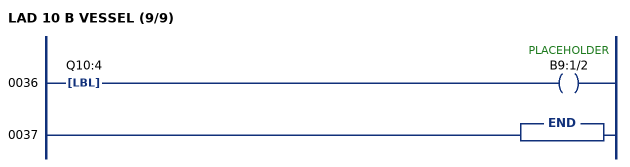
% Rung: 36 %
SOR LBL Q10:4 OTE B9:1/2 EOR
%   B9:1/2  "PLACEHOLDER" %
% Rung: 37 %
SOR END EOR

LADDER 11 "DIGITAL IN"
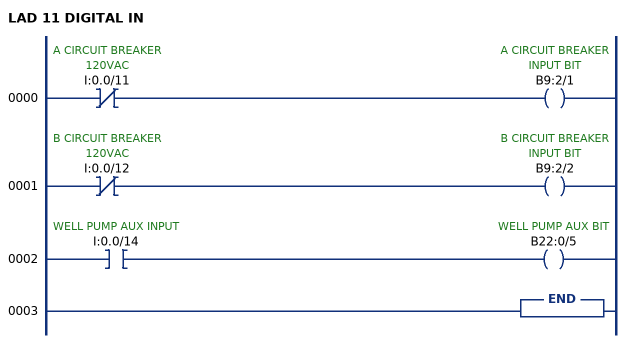
% Rung: 0 %
SOR XIO I:0.0/11 OTE B9:2/1 EOR
%   I:0.0/11  "A CIRCUIT BREAKER 120VAC" %
%   B9:2/1  "A CIRCUIT BREAKER INPUT BIT" %
% Rung: 1 %
SOR XIO I:0.0/12 OTE B9:2/2 EOR
%   I:0.0/12  "B CIRCUIT BREAKER 120VAC" %
%   B9:2/2  "B CIRCUIT BREAKER INPUT BIT" %
% Rung: 2 %
SOR XIC I:0.0/14 OTE B22:0/5 EOR
%   I:0.0/14  "WELL PUMP AUX INPUT" %
%   B22:0/5  "WELL PUMP AUX BIT" %
% Rung: 3 %
SOR END EOR

LADDER 12 "WELL PUMP"
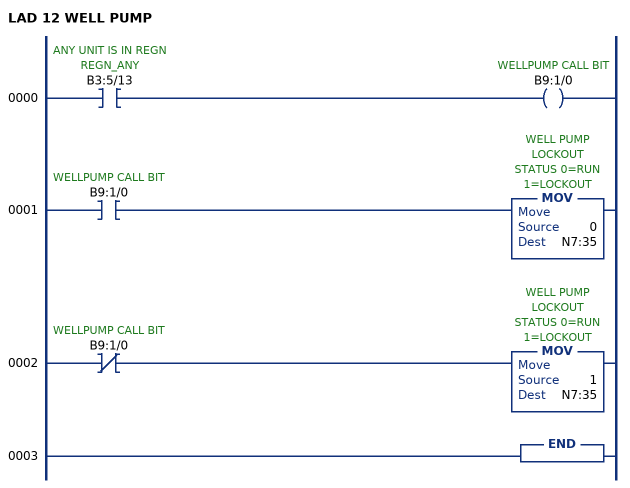
% Rung: 0 %
SOR XIC B3:5/13 OTE B9:1/0 EOR
%   B3:5/13  REGN_ANY  "ANY UNIT IS IN REGN" %
%   B9:1/0  "WELLPUMP CALL BIT" %
% Rung: 1 %
SOR XIC B9:1/0 MOV 0 N7:35 EOR
%   B9:1/0  "WELLPUMP CALL BIT" %
%   N7:35  "WELL PUMP LOCKOUT STATUS 0=RUN 1=LOCKOUT" %
% Rung: 2 %
SOR XIO B9:1/0 MOV 1 N7:35 EOR
%   B9:1/0  "WELLPUMP CALL BIT" %
%   N7:35  "WELL PUMP LOCKOUT STATUS 0=RUN 1=LOCKOUT" %
% Rung: 3 %
SOR END EOR

LADDER 16 "DIGITL OUT"
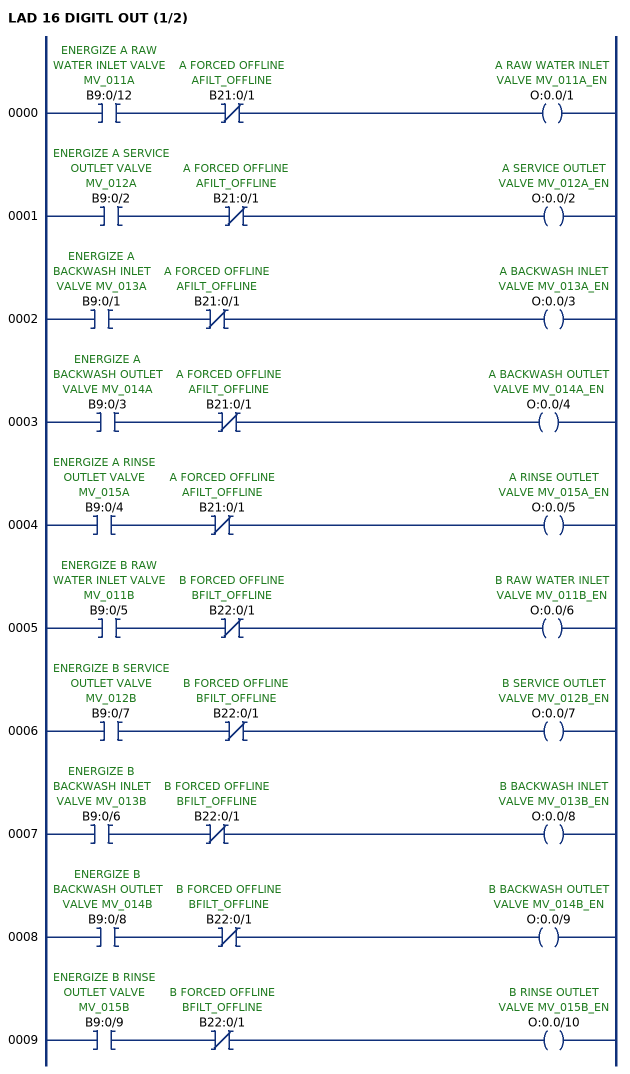
% Rung: 0 %
SOR XIC B9:0/12 XIO B21:0/1 OTE O:0.0/1 EOR
%   B9:0/12  MV_011A  "ENERGIZE A RAW WATER INLET VALVE" %
%   B21:0/1  AFILT_OFFLINE  "A FORCED OFFLINE" %
%   O:0.0/1  MV_011A_EN  "A RAW WATER INLET VALVE" %
% Rung: 1 %
SOR XIC B9:0/2 XIO B21:0/1 OTE O:0.0/2 EOR
%   B9:0/2  MV_012A  "ENERGIZE A SERVICE OUTLET VALVE" %
%   B21:0/1  AFILT_OFFLINE  "A FORCED OFFLINE" %
%   O:0.0/2  MV_012A_EN  "A SERVICE OUTLET VALVE" %
% Rung: 2 %
SOR XIC B9:0/1 XIO B21:0/1 OTE O:0.0/3 EOR
%   B9:0/1  MV_013A  "ENERGIZE A BACKWASH INLET VALVE" %
%   B21:0/1  AFILT_OFFLINE  "A FORCED OFFLINE" %
%   O:0.0/3  MV_013A_EN  "A BACKWASH INLET VALVE" %
% Rung: 3 %
SOR XIC B9:0/3 XIO B21:0/1 OTE O:0.0/4 EOR
%   B9:0/3  MV_014A  "ENERGIZE A BACKWASH OUTLET VALVE" %
%   B21:0/1  AFILT_OFFLINE  "A FORCED OFFLINE" %
%   O:0.0/4  MV_014A_EN  "A BACKWASH OUTLET VALVE" %
% Rung: 4 %
SOR XIC B9:0/4 XIO B21:0/1 OTE O:0.0/5 EOR
%   B9:0/4  MV_015A  "ENERGIZE A RINSE OUTLET VALVE" %
%   B21:0/1  AFILT_OFFLINE  "A FORCED OFFLINE" %
%   O:0.0/5  MV_015A_EN  "A RINSE OUTLET VALVE" %
% Rung: 5 %
SOR XIC B9:0/5 XIO B22:0/1 OTE O:0.0/6 EOR
%   B9:0/5  MV_011B  "ENERGIZE B RAW WATER INLET VALVE" %
%   B22:0/1  BFILT_OFFLINE  "B FORCED OFFLINE" %
%   O:0.0/6  MV_011B_EN  "B RAW WATER INLET VALVE" %
% Rung: 6 %
SOR XIC B9:0/7 XIO B22:0/1 OTE O:0.0/7 EOR
%   B9:0/7  MV_012B  "ENERGIZE B SERVICE OUTLET VALVE" %
%   B22:0/1  BFILT_OFFLINE  "B FORCED OFFLINE" %
%   O:0.0/7  MV_012B_EN  "B SERVICE OUTLET VALVE" %
% Rung: 7 %
SOR XIC B9:0/6 XIO B22:0/1 OTE O:0.0/8 EOR
%   B9:0/6  MV_013B  "ENERGIZE B BACKWASH INLET VALVE" %
%   B22:0/1  BFILT_OFFLINE  "B FORCED OFFLINE" %
%   O:0.0/8  MV_013B_EN  "B BACKWASH INLET VALVE" %
% Rung: 8 %
SOR XIC B9:0/8 XIO B22:0/1 OTE O:0.0/9 EOR
%   B9:0/8  MV_014B  "ENERGIZE B BACKWASH OUTLET VALVE" %
%   B22:0/1  BFILT_OFFLINE  "B FORCED OFFLINE" %
%   O:0.0/9  MV_014B_EN  "B BACKWASH OUTLET VALVE" %
% Rung: 9 %
SOR XIC B9:0/9 XIO B22:0/1 OTE O:0.0/10 EOR
%   B9:0/9  MV_015B  "ENERGIZE B RINSE OUTLET VALVE" %
%   B22:0/1  BFILT_OFFLINE  "B FORCED OFFLINE" %
%   O:0.0/10  MV_015B_EN  "B RINSE OUTLET VALVE" %

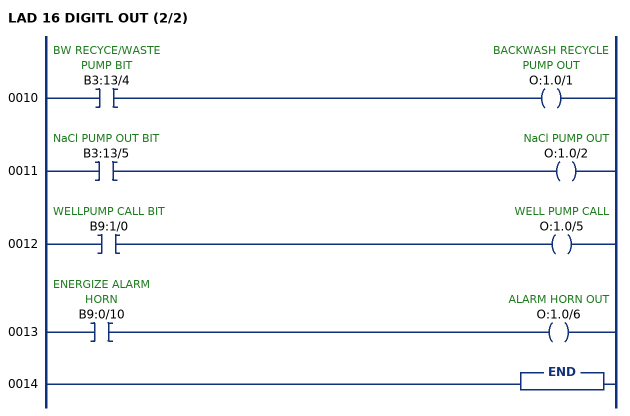
% Rung: 10 %
SOR XIC B3:13/4 OTE O:1.0/1 EOR
%   B3:13/4  "BW RECYCE/WASTE PUMP BIT" %
%   O:1.0/1  "BACKWASH RECYCLE PUMP OUT" %
% Rung: 11 %
SOR XIC B3:13/5 OTE O:1.0/2 EOR
%   B3:13/5  "NaCl PUMP OUT BIT" %
%   O:1.0/2  "NaCl PUMP OUT" %
% Rung: 12 %
SOR XIC B9:1/0 OTE O:1.0/5 EOR
%   B9:1/0  "WELLPUMP CALL BIT" %
%   O:1.0/5  "WELL PUMP CALL" %
% Rung: 13 %
SOR XIC B9:0/10 OTE O:1.0/6 EOR
%   B9:0/10  "ENERGIZE ALARM HORN" %
%   O:1.0/6  "ALARM HORN OUT" %
% Rung: 14 %
SOR END EOR

LADDER 17 "REGEN A"
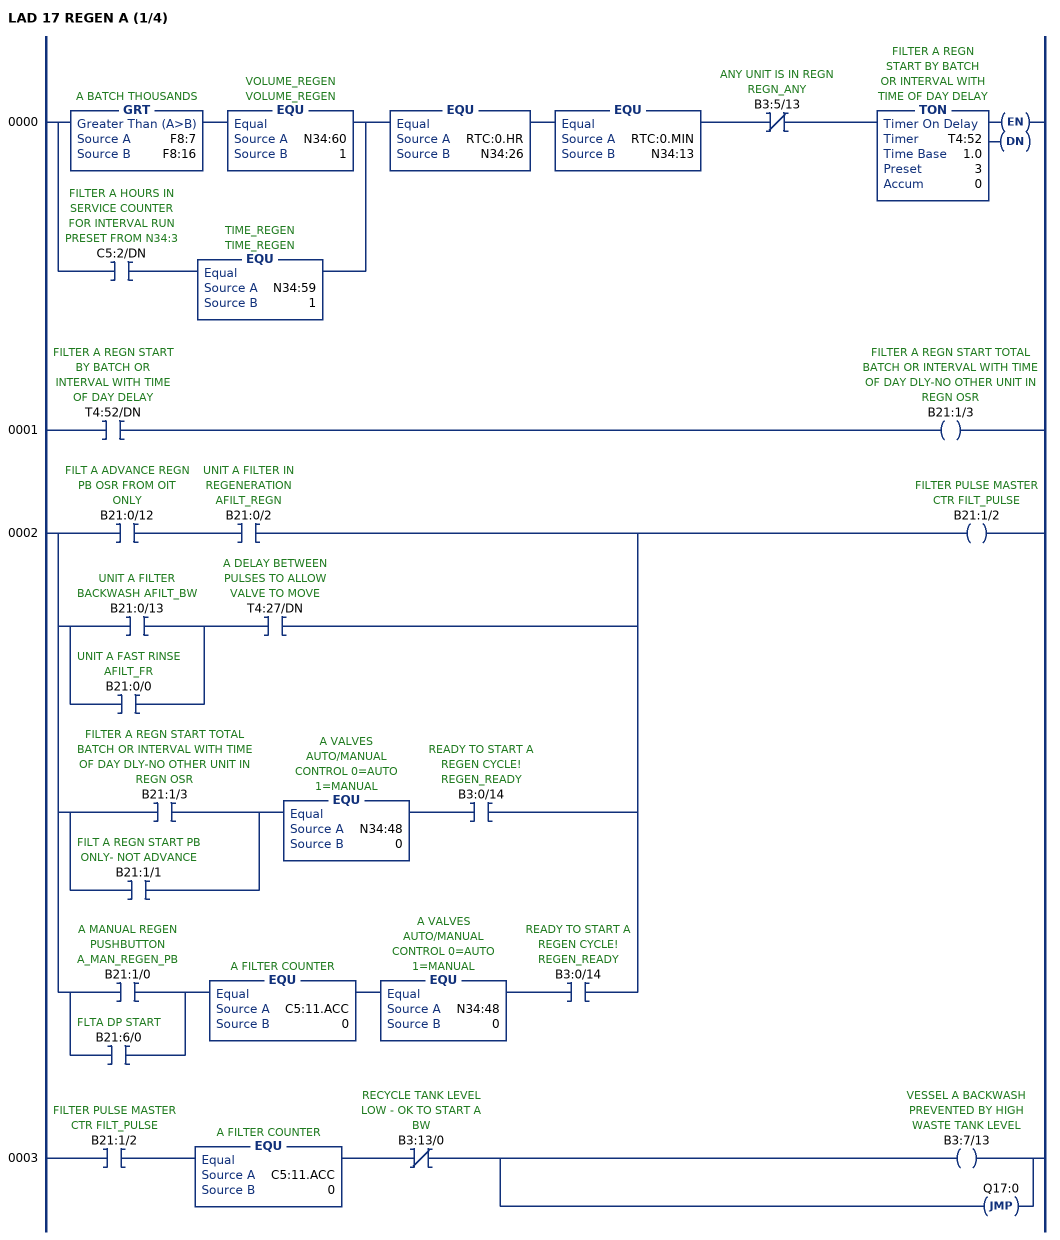
% Rung: 0 %
SOR BST GRT F8:7 F8:16 EQU N34:60 1 NXB XIC C5:2/DN EQU N34:59 1 BND EQU RTC:0.HR N34:26 EQU RTC:0.MIN N34:13 XIO B3:5/13 TON T4:52 1.0 3 0 EOR
%   F8:7  "A BATCH THOUSANDS" %
%   F8:16  T_GAL %
%   N34:60  VOLUME_REGEN  "VOLUME_REGEN" %
%   C5:2  "FILTER A HOURS IN SERVICE COUNTER FOR INTERVAL RUN PRESET FROM N34:3" %
%   N34:59  TIME_REGEN  "TIME_REGEN" %
%   N34:26  "FILTER A HOUR OF DAY TO START SELECT EITHER DUE TO BATCH OR ELAPSED TIME OR DP" %
%   N34:13  "FILTER A MIN OF DAY TO START SELECT EITHER DUE TO BATCH OR ELAPSED TIME" %
%   B3:5/13  REGN_ANY  "ANY UNIT IS IN REGN" %
%   T4:52  "FILTER A REGN START BY BATCH OR INTERVAL WITH TIME OF DAY DELAY" %
% Rung: 1 %
SOR XIC T4:52/DN OTE B21:1/3 EOR
%   T4:52  "FILTER A REGN START BY BATCH OR INTERVAL WITH TIME OF DAY DELAY" %
%   B21:1/3  "FILTER A REGN START TOTAL BATCH OR INTERVAL WITH TIME OF DAY DLY-NO OTHER UNIT IN REGN OSR" %
% Rung: 2 %
SOR BST BST BST XIC B21:0/12 XIC B21:0/2 NXB BST XIC B21:0/13 NXB XIC B21:0/0 BND XIC T4:27/DN BND NXB BST XIC B21:1/3 NXB XIC B21:1/1 BND EQU N34:48 0 XIC B3:0/14 BND NXB BST XIC B21:1/0 NXB XIC B21:6/0 BND EQU C5:11.ACC 0 EQU N34:48 0 XIC B3:0/14 BND OTE B21:1/2 EOR
%   B21:0/12  "FILT A ADVANCE REGN PB OSR FROM OIT ONLY" %
%   B21:0/2  AFILT_REGN  "UNIT A FILTER IN REGENERATION" %
%   B21:0/13  AFILT_BW  "UNIT A FILTER BACKWASH" %
%   B21:0/0  AFILT_FR  "UNIT A FAST RINSE" %
%   T4:27  "A DELAY BETWEEN PULSES TO ALLOW VALVE TO MOVE" %
%   B21:1/3  "FILTER A REGN START TOTAL BATCH OR INTERVAL WITH TIME OF DAY DLY-NO OTHER UNIT IN REGN OSR" %
%   B21:1/1  "FILT A REGN START PB ONLY- NOT ADVANCE" %
%   N34:48  "A VALVES AUTO/MANUAL CONTROL 0=AUTO 1=MANUAL" %
%   B3:0/14  REGEN_READY  "READY TO START A REGEN CYCLE!" %
%   B21:1/0  A_MAN_REGEN_PB  "A MANUAL REGEN PUSHBUTTON" %
%   B21:6/0  "FLTA DP START" %
%   C5:11.ACC  "A FILTER COUNTER" %
%   B21:1/2  FILT_PULSE  "FILTER PULSE MASTER CTR" %
% Rung: 3 %
SOR XIC B21:1/2 EQU C5:11.ACC 0 XIO B3:13/0 BST OTE B3:7/13 NXB JMP Q17:0 BND EOR
%   B21:1/2  FILT_PULSE  "FILTER PULSE MASTER CTR" %
%   C5:11.ACC  "A FILTER COUNTER" %
%   B3:13/0  "RECYCLE TANK LEVEL LOW - OK TO START A BW" %
%   B3:7/13  "VESSEL A BACKWASH PREVENTED BY HIGH WASTE TANK LEVEL" %

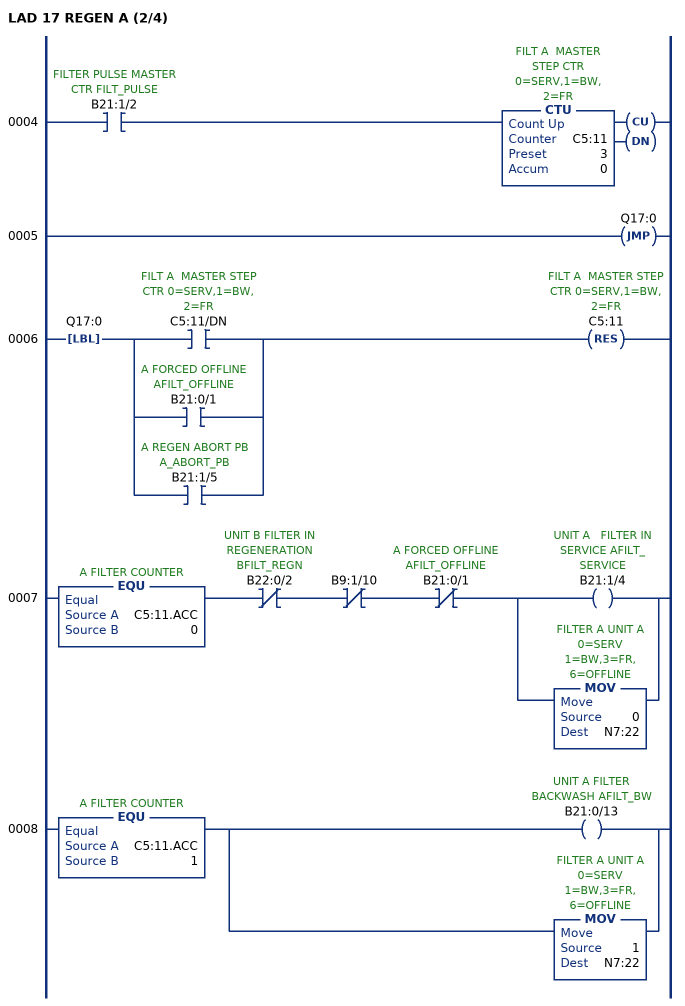
% Rung: 4 %
SOR XIC B21:1/2 CTU C5:11 3 0 EOR
%   B21:1/2  FILT_PULSE  "FILTER PULSE MASTER CTR" %
%   C5:11  "FILT A  MASTER STEP CTR 0=SERV,1=BW,2=FR" %
% Rung: 5 %
SOR JMP Q17:0 EOR
% Rung: 6 %
SOR LBL Q17:0 BST XIC C5:11/DN NXB XIC B21:0/1 NXB XIC B21:1/5 BND RES C5:11 EOR
%   C5:11  "FILT A  MASTER STEP CTR 0=SERV,1=BW,2=FR" %
%   B21:0/1  AFILT_OFFLINE  "A FORCED OFFLINE" %
%   B21:1/5  A_ABORT_PB  "A REGEN ABORT PB" %
% Rung: 7 %
SOR EQU C5:11.ACC 0 XIO B22:0/2 XIO B9:1/10 XIO B21:0/1 BST OTE B21:1/4 NXB MOV 0 N7:22 BND EOR
%   C5:11.ACC  "A FILTER COUNTER" %
%   B22:0/2  BFILT_REGN  "UNIT B FILTER IN REGENERATION" %
%   B21:0/1  AFILT_OFFLINE  "A FORCED OFFLINE" %
%   B21:1/4  AFILT_SERVICE  "UNIT A   FILTER IN SERVICE" %
%   N7:22  "FILTER A UNIT A 0=SERV 1=BW,3=FR,6=OFFLINE" %
% Rung: 8 %
SOR EQU C5:11.ACC 1 BST OTE B21:0/13 NXB MOV 1 N7:22 BND EOR
%   C5:11.ACC  "A FILTER COUNTER" %
%   B21:0/13  AFILT_BW  "UNIT A FILTER BACKWASH" %
%   N7:22  "FILTER A UNIT A 0=SERV 1=BW,3=FR,6=OFFLINE" %

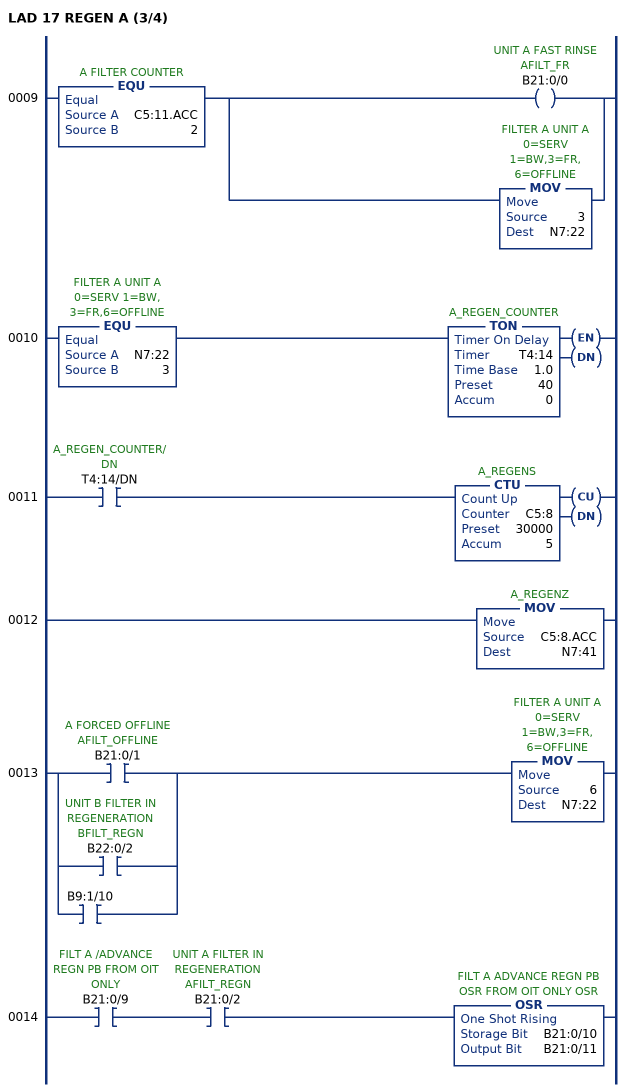
% Rung: 9 %
SOR EQU C5:11.ACC 2 BST OTE B21:0/0 NXB MOV 3 N7:22 BND EOR
%   C5:11.ACC  "A FILTER COUNTER" %
%   B21:0/0  AFILT_FR  "UNIT A FAST RINSE" %
%   N7:22  "FILTER A UNIT A 0=SERV 1=BW,3=FR,6=OFFLINE" %
% Rung: 10 %
SOR EQU N7:22 3 TON T4:14 1.0 40 0 EOR
%   N7:22  "FILTER A UNIT A 0=SERV 1=BW,3=FR,6=OFFLINE" %
%   T4:14  A_REGEN_COUNTER %
% Rung: 11 %
SOR XIC T4:14/DN CTU C5:8 30000 5 EOR
%   T4:14  A_REGEN_COUNTER %
%   C5:8  "A_REGENS" %
% Rung: 12 %
SOR MOV C5:8.ACC N7:41 EOR
%   C5:8  "A_REGENS" %
%   N7:41  A_REGENZ %
% Rung: 13 %
SOR BST XIC B21:0/1 NXB XIC B22:0/2 NXB XIC B9:1/10 BND MOV 6 N7:22 EOR
%   B21:0/1  AFILT_OFFLINE  "A FORCED OFFLINE" %
%   B22:0/2  BFILT_REGN  "UNIT B FILTER IN REGENERATION" %
%   N7:22  "FILTER A UNIT A 0=SERV 1=BW,3=FR,6=OFFLINE" %
% Rung: 14 %
SOR XIC B21:0/9 XIC B21:0/2 OSR B21:0/10 B21:0/11 EOR
%   B21:0/9  "FILT A /ADVANCE REGN PB FROM OIT ONLY" %
%   B21:0/2  AFILT_REGN  "UNIT A FILTER IN REGENERATION" %
%   B21:0/10  "FILT A ADVANCE REGN PB OSR FROM OIT ONLY OSR" %
%   B21:0/11  "FILT A START/ADVANCE REGN PB OSR FROM OIT ONLY OSR" %

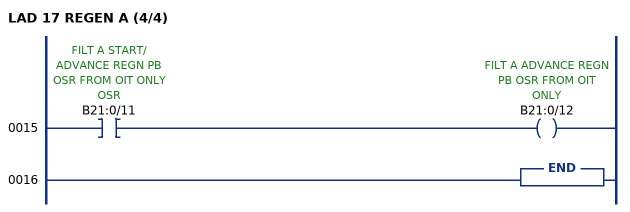
% Rung: 15 %
SOR XIC B21:0/11 OTE B21:0/12 EOR
%   B21:0/11  "FILT A START/ADVANCE REGN PB OSR FROM OIT ONLY OSR" %
%   B21:0/12  "FILT A ADVANCE REGN PB OSR FROM OIT ONLY" %
% Rung: 16 %
SOR END EOR

LADDER 18 "REGEN B"
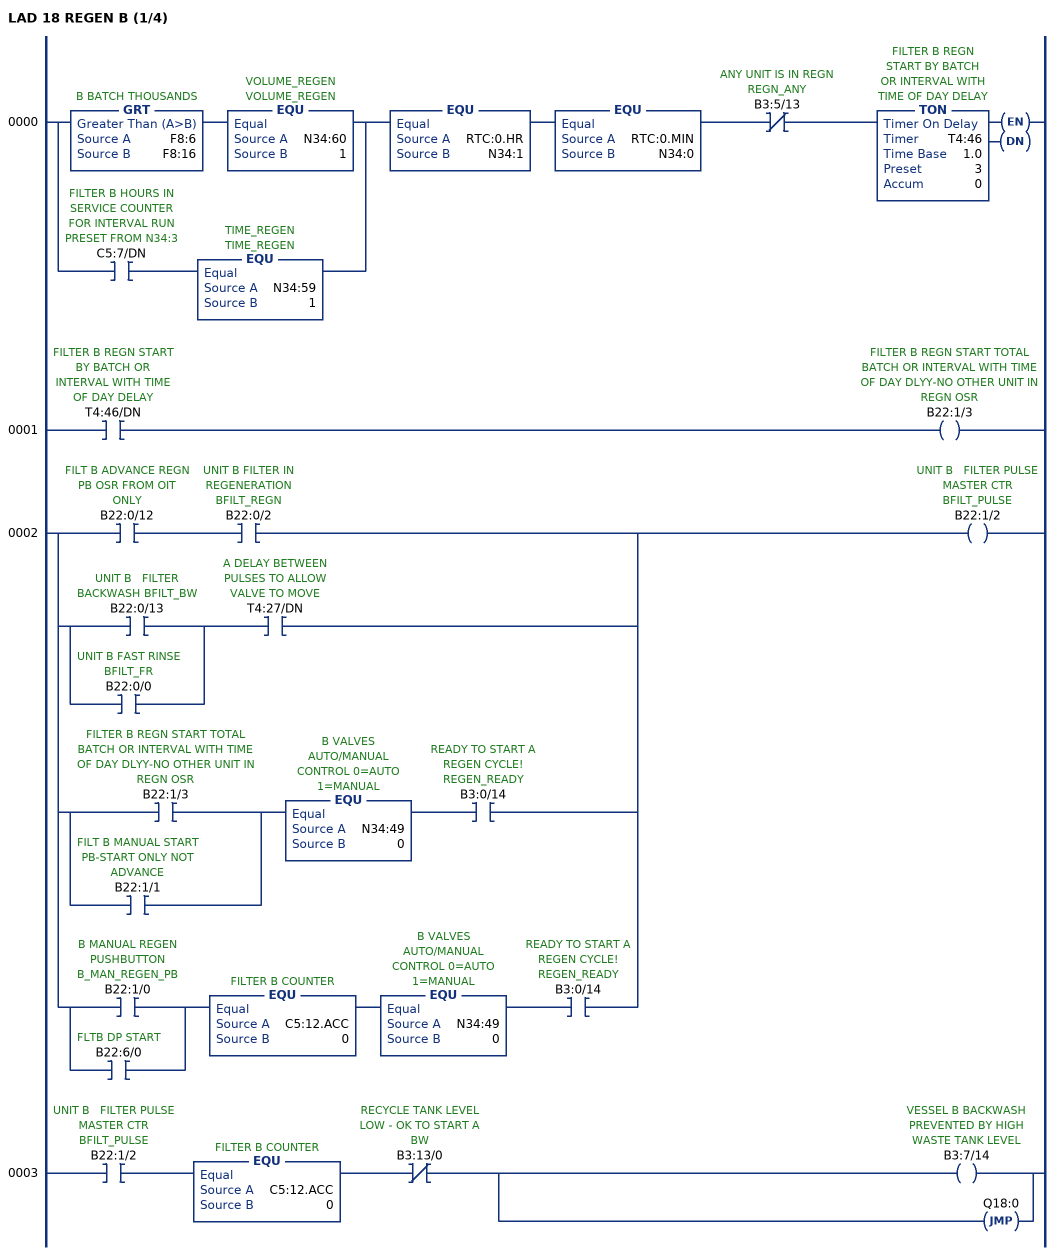
% Rung: 0 %
SOR BST GRT F8:6 F8:16 EQU N34:60 1 NXB XIC C5:7/DN EQU N34:59 1 BND EQU RTC:0.HR N34:1 EQU RTC:0.MIN N34:0 XIO B3:5/13 TON T4:46 1.0 3 0 EOR
%   F8:6  "B BATCH THOUSANDS" %
%   F8:16  T_GAL %
%   N34:60  VOLUME_REGEN  "VOLUME_REGEN" %
%   C5:7  "FILTER B HOURS IN SERVICE COUNTER FOR INTERVAL RUN PRESET FROM N34:3" %
%   N34:59  TIME_REGEN  "TIME_REGEN" %
%   N34:1  "FILTER B HOUR OF DAY TO START SELECT EITHER DUE TO BATCH OR ELAPSED TIME OR DP" %
%   N34:0  "FILTER B MIN OF DAY TO START SELECT EITHER DUE TO BATCH OR ELAPSED TIME" %
%   B3:5/13  REGN_ANY  "ANY UNIT IS IN REGN" %
%   T4:46  "FILTER B REGN START BY BATCH OR INTERVAL WITH TIME OF DAY DELAY" %
% Rung: 1 %
SOR XIC T4:46/DN OTE B22:1/3 EOR
%   T4:46  "FILTER B REGN START BY BATCH OR INTERVAL WITH TIME OF DAY DELAY" %
%   B22:1/3  "FILTER B REGN START TOTAL BATCH OR INTERVAL WITH TIME OF DAY DLYY-NO OTHER UNIT IN REGN OSR" %
% Rung: 2 %
SOR BST BST BST XIC B22:0/12 XIC B22:0/2 NXB BST XIC B22:0/13 NXB XIC B22:0/0 BND XIC T4:27/DN BND NXB BST XIC B22:1/3 NXB XIC B22:1/1 BND EQU N34:49 0 XIC B3:0/14 BND NXB BST XIC B22:1/0 NXB XIC B22:6/0 BND EQU C5:12.ACC 0 EQU N34:49 0 XIC B3:0/14 BND OTE B22:1/2 EOR
%   B22:0/12  "FILT B ADVANCE REGN PB OSR FROM OIT ONLY" %
%   B22:0/2  BFILT_REGN  "UNIT B FILTER IN REGENERATION" %
%   B22:0/13  BFILT_BW  "UNIT B   FILTER BACKWASH" %
%   B22:0/0  BFILT_FR  "UNIT B FAST RINSE" %
%   T4:27  "A DELAY BETWEEN PULSES TO ALLOW VALVE TO MOVE" %
%   B22:1/3  "FILTER B REGN START TOTAL BATCH OR INTERVAL WITH TIME OF DAY DLYY-NO OTHER UNIT IN REGN OSR" %
%   B22:1/1  "FILT B MANUAL START PB-START ONLY NOT ADVANCE" %
%   N34:49  "B VALVES AUTO/MANUAL CONTROL 0=AUTO 1=MANUAL" %
%   B3:0/14  REGEN_READY  "READY TO START A REGEN CYCLE!" %
%   B22:1/0  B_MAN_REGEN_PB  "B MANUAL REGEN PUSHBUTTON" %
%   B22:6/0  "FLTB DP START" %
%   C5:12.ACC  "FILTER B COUNTER" %
%   B22:1/2  BFILT_PULSE  "UNIT B   FILTER PULSE MASTER CTR" %
% Rung: 3 %
SOR XIC B22:1/2 EQU C5:12.ACC 0 XIO B3:13/0 BST OTE B3:7/14 NXB JMP Q18:0 BND EOR
%   B22:1/2  BFILT_PULSE  "UNIT B   FILTER PULSE MASTER CTR" %
%   C5:12.ACC  "FILTER B COUNTER" %
%   B3:13/0  "RECYCLE TANK LEVEL LOW - OK TO START A BW" %
%   B3:7/14  "VESSEL B BACKWASH PREVENTED BY HIGH WASTE TANK LEVEL" %

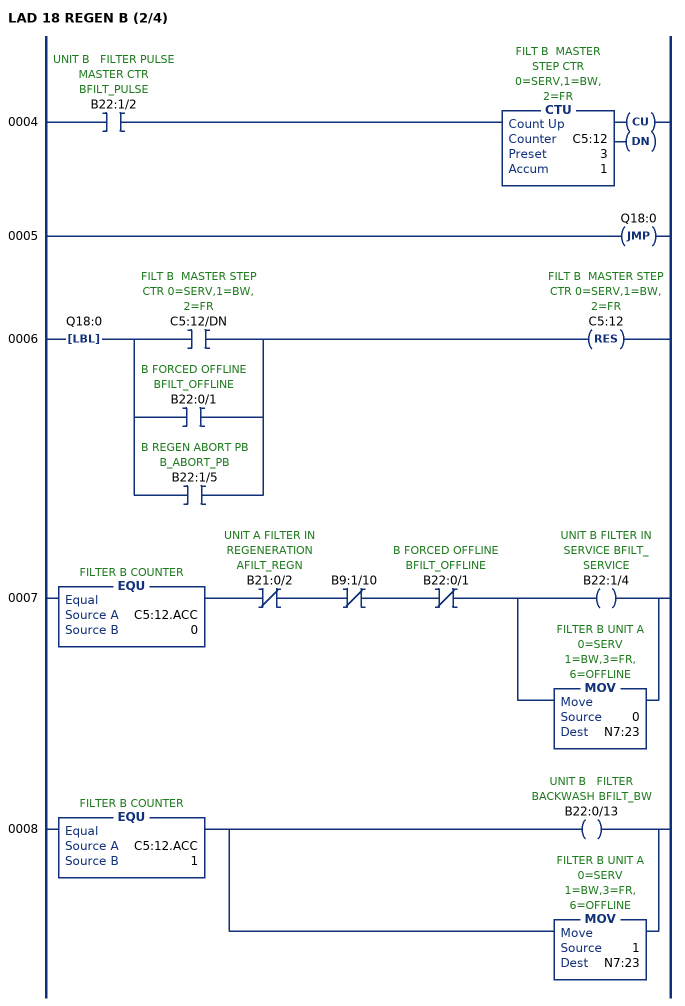
% Rung: 4 %
SOR XIC B22:1/2 CTU C5:12 3 1 EOR
%   B22:1/2  BFILT_PULSE  "UNIT B   FILTER PULSE MASTER CTR" %
%   C5:12  "FILT B  MASTER STEP CTR 0=SERV,1=BW,2=FR" %
% Rung: 5 %
SOR JMP Q18:0 EOR
% Rung: 6 %
SOR LBL Q18:0 BST XIC C5:12/DN NXB XIC B22:0/1 NXB XIC B22:1/5 BND RES C5:12 EOR
%   C5:12  "FILT B  MASTER STEP CTR 0=SERV,1=BW,2=FR" %
%   B22:0/1  BFILT_OFFLINE  "B FORCED OFFLINE" %
%   B22:1/5  B_ABORT_PB  "B REGEN ABORT PB" %
% Rung: 7 %
SOR EQU C5:12.ACC 0 XIO B21:0/2 XIO B9:1/10 XIO B22:0/1 BST OTE B22:1/4 NXB MOV 0 N7:23 BND EOR
%   C5:12.ACC  "FILTER B COUNTER" %
%   B21:0/2  AFILT_REGN  "UNIT A FILTER IN REGENERATION" %
%   B22:0/1  BFILT_OFFLINE  "B FORCED OFFLINE" %
%   B22:1/4  BFILT_SERVICE  "UNIT B FILTER IN SERVICE" %
%   N7:23  "FILTER B UNIT A 0=SERV 1=BW,3=FR,6=OFFLINE" %
% Rung: 8 %
SOR EQU C5:12.ACC 1 BST OTE B22:0/13 NXB MOV 1 N7:23 BND EOR
%   C5:12.ACC  "FILTER B COUNTER" %
%   B22:0/13  BFILT_BW  "UNIT B   FILTER BACKWASH" %
%   N7:23  "FILTER B UNIT A 0=SERV 1=BW,3=FR,6=OFFLINE" %

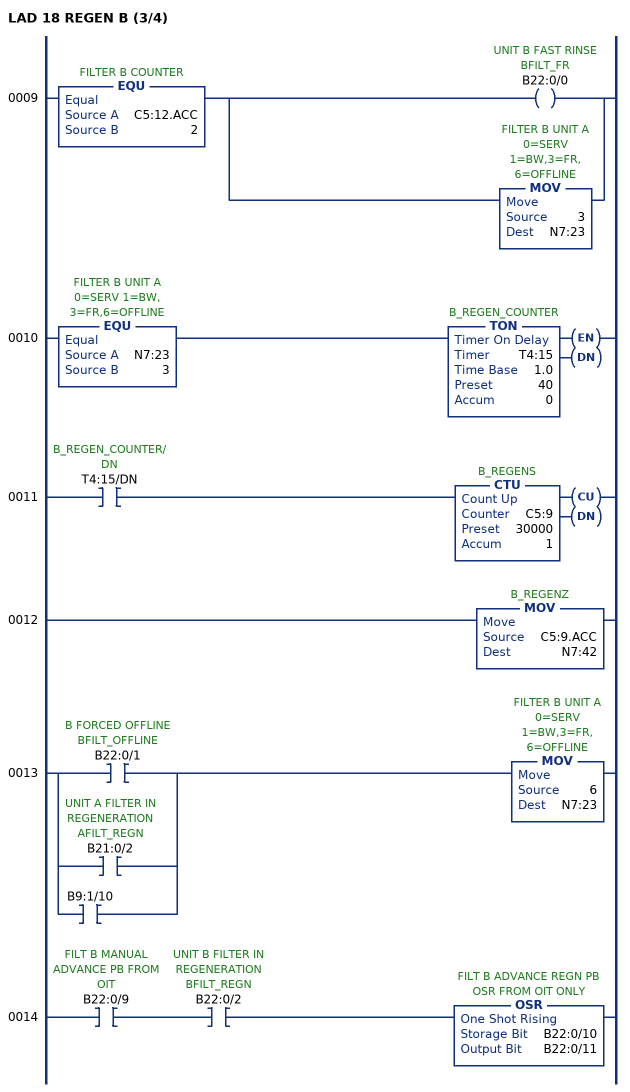
% Rung: 9 %
SOR EQU C5:12.ACC 2 BST OTE B22:0/0 NXB MOV 3 N7:23 BND EOR
%   C5:12.ACC  "FILTER B COUNTER" %
%   B22:0/0  BFILT_FR  "UNIT B FAST RINSE" %
%   N7:23  "FILTER B UNIT A 0=SERV 1=BW,3=FR,6=OFFLINE" %
% Rung: 10 %
SOR EQU N7:23 3 TON T4:15 1.0 40 0 EOR
%   N7:23  "FILTER B UNIT A 0=SERV 1=BW,3=FR,6=OFFLINE" %
%   T4:15  B_REGEN_COUNTER %
% Rung: 11 %
SOR XIC T4:15/DN CTU C5:9 30000 1 EOR
%   T4:15  B_REGEN_COUNTER %
%   C5:9  "B_REGENS" %
% Rung: 12 %
SOR MOV C5:9.ACC N7:42 EOR
%   C5:9  "B_REGENS" %
%   N7:42  B_REGENZ %
% Rung: 13 %
SOR BST XIC B22:0/1 NXB XIC B21:0/2 NXB XIC B9:1/10 BND MOV 6 N7:23 EOR
%   B22:0/1  BFILT_OFFLINE  "B FORCED OFFLINE" %
%   B21:0/2  AFILT_REGN  "UNIT A FILTER IN REGENERATION" %
%   N7:23  "FILTER B UNIT A 0=SERV 1=BW,3=FR,6=OFFLINE" %
% Rung: 14 %
SOR XIC B22:0/9 XIC B22:0/2 OSR B22:0/10 B22:0/11 EOR
%   B22:0/9  "FILT B MANUAL ADVANCE PB FROM OIT" %
%   B22:0/2  BFILT_REGN  "UNIT B FILTER IN REGENERATION" %
%   B22:0/10  "FILT B ADVANCE REGN PB OSR FROM OIT ONLY" %
%   B22:0/11  "FILT B /ADVANCE REGN PB OSR FROM OIT ONLY" %

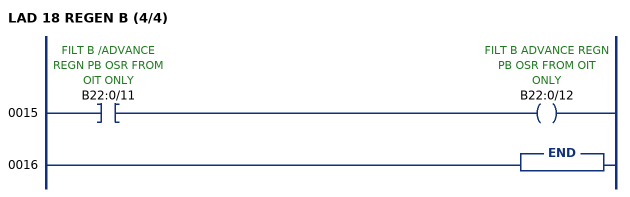
% Rung: 15 %
SOR XIC B22:0/11 OTE B22:0/12 EOR
%   B22:0/11  "FILT B /ADVANCE REGN PB OSR FROM OIT ONLY" %
%   B22:0/12  "FILT B ADVANCE REGN PB OSR FROM OIT ONLY" %
% Rung: 16 %
SOR END EOR

LADDER 19 "RECYCLE"
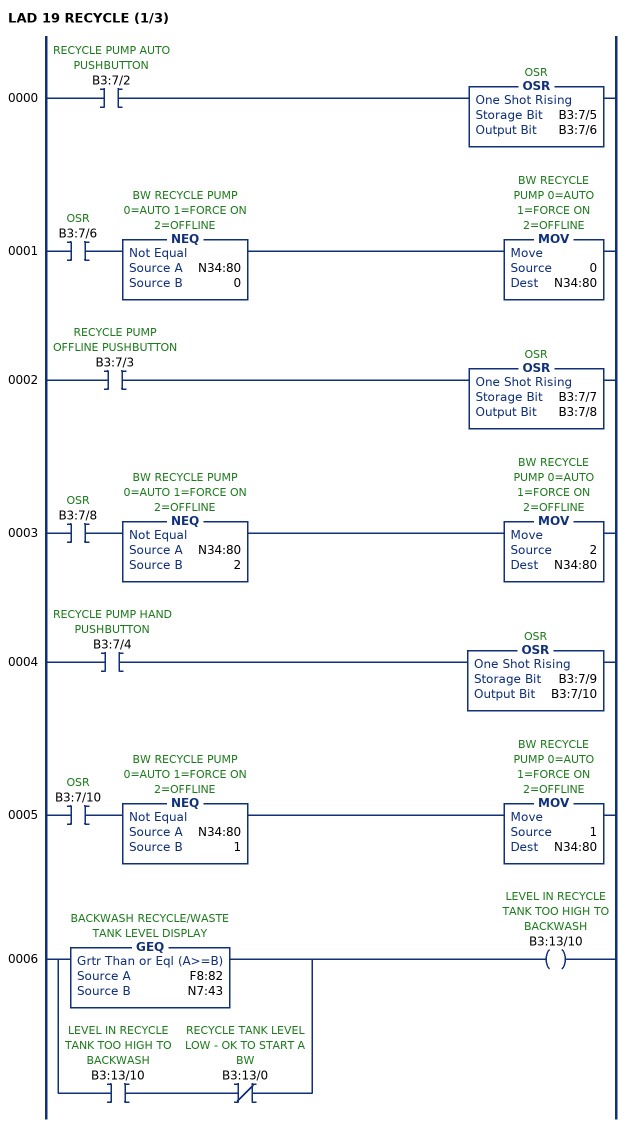
% Rung: 0 %
SOR XIC B3:7/2 OSR B3:7/5 B3:7/6 EOR
%   B3:7/2  "RECYCLE PUMP AUTO PUSHBUTTON" %
%   B3:7/5  "OSR" %
%   B3:7/6  "OSR" %
% Rung: 1 %
SOR XIC B3:7/6 NEQ N34:80 0 MOV 0 N34:80 EOR
%   B3:7/6  "OSR" %
%   N34:80  "BW RECYCLE PUMP 0=AUTO 1=FORCE ON 2=OFFLINE" %
% Rung: 2 %
SOR XIC B3:7/3 OSR B3:7/7 B3:7/8 EOR
%   B3:7/3  "RECYCLE PUMP OFFLINE PUSHBUTTON" %
%   B3:7/7  "OSR" %
%   B3:7/8  "OSR" %
% Rung: 3 %
SOR XIC B3:7/8 NEQ N34:80 2 MOV 2 N34:80 EOR
%   B3:7/8  "OSR" %
%   N34:80  "BW RECYCLE PUMP 0=AUTO 1=FORCE ON 2=OFFLINE" %
% Rung: 4 %
SOR XIC B3:7/4 OSR B3:7/9 B3:7/10 EOR
%   B3:7/4  "RECYCLE PUMP HAND PUSHBUTTON" %
%   B3:7/9  "OSR" %
%   B3:7/10  "OSR" %
% Rung: 5 %
SOR XIC B3:7/10 NEQ N34:80 1 MOV 1 N34:80 EOR
%   B3:7/10  "OSR" %
%   N34:80  "BW RECYCLE PUMP 0=AUTO 1=FORCE ON 2=OFFLINE" %
% Rung: 6 %
SOR BST GEQ F8:82 N7:43 NXB XIC B3:13/10 XIO B3:13/0 BND OTE B3:13/10 EOR
%   F8:82  "BACKWASH RECYCLE/WASTE TANK LEVEL DISPLAY" %
%   N7:43  "LEVEL IN BW WASTE TANK TO PREVENT A REGN START- TANK IS TOO HIGH TO ACCEPT BW WASTE  (HI)" %
%   B3:13/10  "LEVEL IN RECYCLE TANK TOO HIGH TO BACKWASH" %
%   B3:13/0  "RECYCLE TANK LEVEL LOW - OK TO START A BW" %

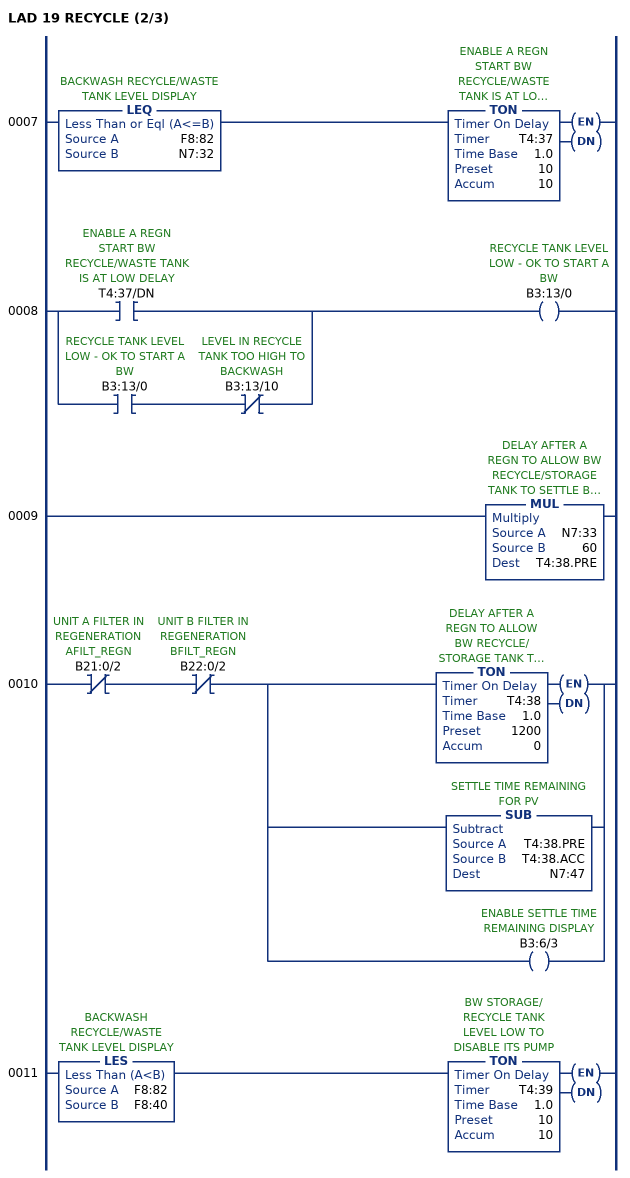
% Rung: 7 %
SOR LEQ F8:82 N7:32 TON T4:37 1.0 10 10 EOR
%   F8:82  "BACKWASH RECYCLE/WASTE TANK LEVEL DISPLAY" %
%   N7:32  "LOW LEVEL ENTRY TO ENABLE A BW START.IF LVL IS NOT LOW THEN A BW MIGHT OVERFLOW TANK." %
%   T4:37  "ENABLE A REGN START BW RECYCLE/WASTE TANK IS AT LOW DELAY" %
% Rung: 8 %
SOR BST XIC T4:37/DN NXB XIC B3:13/0 XIO B3:13/10 BND OTE B3:13/0 EOR
%   T4:37  "ENABLE A REGN START BW RECYCLE/WASTE TANK IS AT LOW DELAY" %
%   B3:13/0  "RECYCLE TANK LEVEL LOW - OK TO START A BW" %
%   B3:13/10  "LEVEL IN RECYCLE TANK TOO HIGH TO BACKWASH" %
% Rung: 9 %
SOR MUL N7:33 60 T4:38.PRE EOR
%   N7:33  "DELAY AFTER A REGN END TO ALLOW SETTLING IN TANK B4 STARTING RECLAIM PUMP" %
%   T4:38  "DELAY AFTER A REGN TO ALLOW BW RECYCLE/STORAGE TANK TO SETTLE B4 TURNING ON PMP TO EMPTY" %
% Rung: 10 %
SOR XIO B21:0/2 XIO B22:0/2 BST TON T4:38 1.0 1200 0 NXB SUB T4:38.PRE T4:38.ACC N7:47 NXB OTE B3:6/3 BND EOR
%   B21:0/2  AFILT_REGN  "UNIT A FILTER IN REGENERATION" %
%   B22:0/2  BFILT_REGN  "UNIT B FILTER IN REGENERATION" %
%   T4:38  "DELAY AFTER A REGN TO ALLOW BW RECYCLE/STORAGE TANK TO SETTLE B4 TURNING ON PMP TO EMPTY" %
%   N7:47  "SETTLE TIME REMAINING FOR PV" %
%   B3:6/3  "ENABLE SETTLE TIME REMAINING DISPLAY" %
% Rung: 11 %
SOR LES F8:82 F8:40 TON T4:39 1.0 10 10 EOR
%   F8:82  "BACKWASH RECYCLE/WASTE TANK LEVEL DISPLAY" %
%   F8:40  "TANK LO" %
%   T4:39  "BW STORAGE/RECYCLE TANK LEVEL LOW TO DISABLE ITS PUMP" %

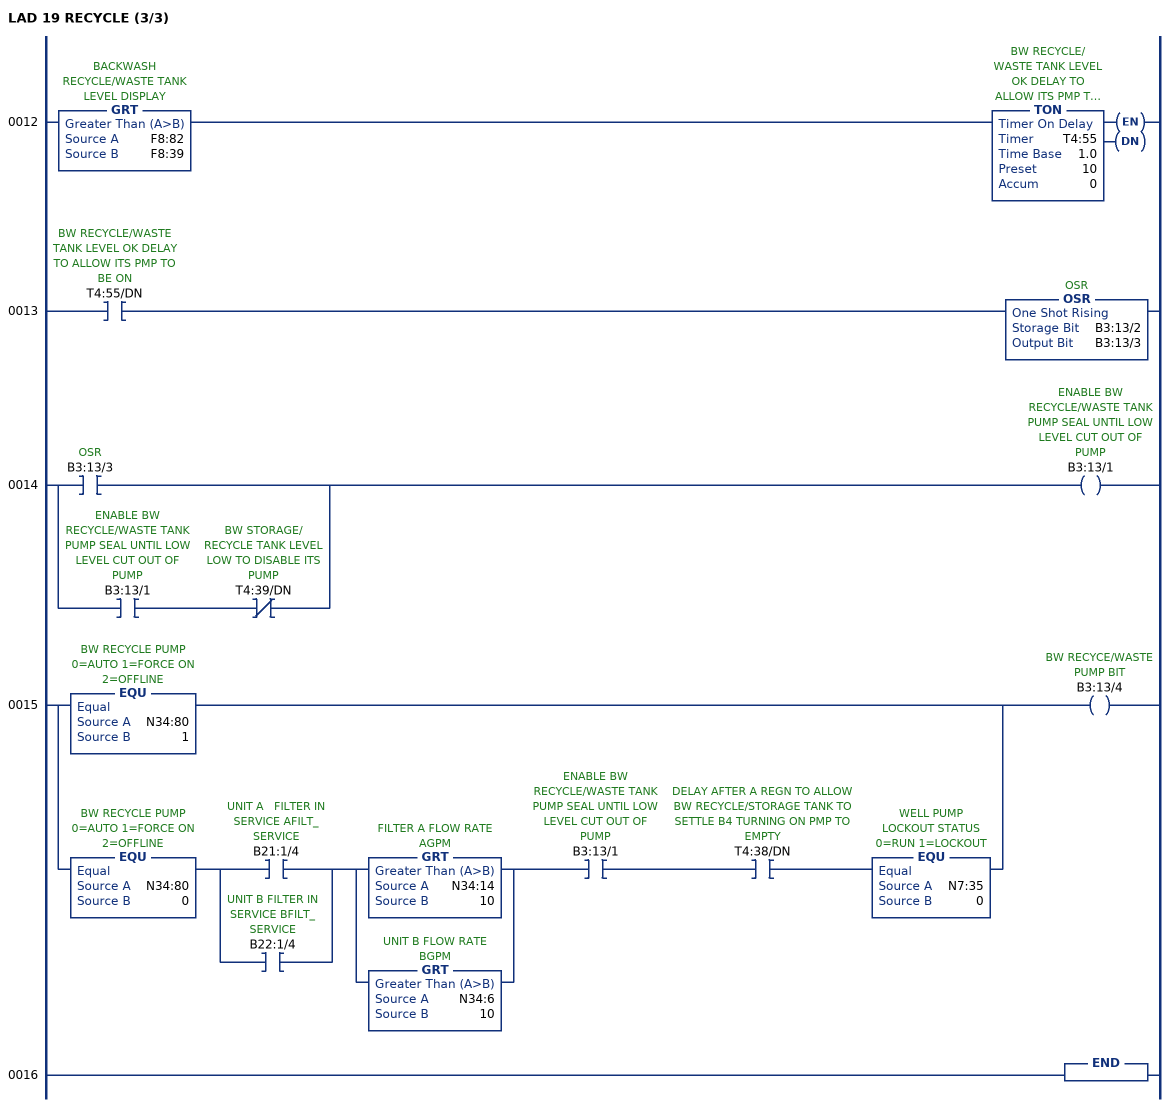
% Rung: 12 %
SOR GRT F8:82 F8:39 TON T4:55 1.0 10 0 EOR
%   F8:82  "BACKWASH RECYCLE/WASTE TANK LEVEL DISPLAY" %
%   F8:39  "TANK HI" %
%   T4:55  "BW RECYCLE/WASTE TANK LEVEL OK DELAY TO ALLOW ITS PMP TO BE ON" %
% Rung: 13 %
SOR XIC T4:55/DN OSR B3:13/2 B3:13/3 EOR
%   T4:55  "BW RECYCLE/WASTE TANK LEVEL OK DELAY TO ALLOW ITS PMP TO BE ON" %
%   B3:13/2  "OSR" %
%   B3:13/3  "OSR" %
% Rung: 14 %
SOR BST XIC B3:13/3 NXB XIC B3:13/1 XIO T4:39/DN BND OTE B3:13/1 EOR
%   B3:13/3  "OSR" %
%   B3:13/1  "ENABLE BW RECYCLE/WASTE TANK PUMP SEAL UNTIL LOW LEVEL CUT OUT OF PUMP" %
%   T4:39  "BW STORAGE/RECYCLE TANK LEVEL LOW TO DISABLE ITS PUMP" %
% Rung: 15 %
SOR BST EQU N34:80 1 NXB EQU N34:80 0 BST XIC B21:1/4 NXB XIC B22:1/4 BND BST GRT N34:14 10 NXB GRT N34:6 10 BND XIC B3:13/1 XIC T4:38/DN EQU N7:35 0 BND OTE B3:13/4 EOR
%   N34:80  "BW RECYCLE PUMP 0=AUTO 1=FORCE ON 2=OFFLINE" %
%   B21:1/4  AFILT_SERVICE  "UNIT A   FILTER IN SERVICE" %
%   B22:1/4  BFILT_SERVICE  "UNIT B FILTER IN SERVICE" %
%   N34:14  AGPM  "FILTER A FLOW RATE" %
%   N34:6  BGPM  "UNIT B FLOW RATE" %
%   B3:13/1  "ENABLE BW RECYCLE/WASTE TANK PUMP SEAL UNTIL LOW LEVEL CUT OUT OF PUMP" %
%   T4:38  "DELAY AFTER A REGN TO ALLOW BW RECYCLE/STORAGE TANK TO SETTLE B4 TURNING ON PMP TO EMPTY" %
%   N7:35  "WELL PUMP LOCKOUT STATUS 0=RUN 1=LOCKOUT" %
%   B3:13/4  "BW RECYCE/WASTE PUMP BIT" %
% Rung: 16 %
SOR END EOR

OTHER DOCUMENTED ADDRESSES
  1F  
  B3:0/15  "RESET SV-800-09 DUE TO LOW CO2 PSI"
  B3:1/0  "WELL PUMP ENABLED DISPLAY ON PV"
  B3:2/13  "FLOW SENSOR A PULS OSR"
  B3:2/14  "FLOW SENSOR A PULS OSR"
  B3:3/0  "FLOW SENSOR B PULSE OSR"
  B3:3/1  "FLOW SENSOR B PULSE OSR"
  B3:3/15  WP_LO
  B3:4/10  "DP CHOSEN AND DELAY DONE OSR"
  B3:4/11  "DP CHOSEN AND DELAY DONE OSR"
  B3:4/15  "ANY UNIT IN FR PLUS NUMBER OF REGN COUNTERS FOR TRACKING SEQUENTIAL RERN MEM OSR"
  B3:6/14  "A PULS CTR OSR"
  B3:7/0  "B PULS CTR OSR"
  B3:7/1  "B PULS CTR OSR"
  B3:8/6  "OSR"
  B3:8/7  "OSR"
  B3:9/3  "MODULATING IS BEING FORCED"
  B3:10/1  "C FILT PULS OSR"
  B3:10/2  "C FILT PULS OSR"
  B3:10/3  "FILT A MULTIPORT VALVE OUTPUT FOR ADV PB LOCKOUT LOGIC"
  B3:10/4  "FILT A MULTIPORT VALVE OUTPUT FOR ADV PB LOCKOUT LOGIC"
  B3:10/6  "FILT B MULTIPORT VALVE OUTPUT FOR ADV PB LOCKOUT LOGIC"
  B3:10/7  "FILT B MULTIPORT VALVE OUTPUT FOR ADV PB LOCKOUT LOGIC"
  B3:10/8  "FILT B MULTIPORT VALVE OUTPUT FOR ADV PB LOCKOUT LOGIC DISPLAY"
  B3:10/9  "FILT C MULTIPORT VALVE OUTPUT FOR ADV PB LOCKOUT LOGIC"
  B3:10/10  "FILT C MULTIPORT VALVE OUTPUT FOR ADV PB LOCKOUT LOGIC"
  B3:10/11  "FILT C MULTIPORT VALVE OUTPUT FOR ADV PB LOCKOUT LOGIC DISPLAY"
  B3:10/12  "FV101A VLV INDICATOR ON PV"
  B3:10/13  "FV102A VLV INDICATOR ON PV"
  B3:10/14  "FV101B VLV INDICATOR ON PV"
  B3:10/15  "FV102B VLV INDICATOR ON PV"
  B3:11/0  "FV101C VLV INDICATOR ON PV"
  B3:11/1  "FV102C VLV INDICATOR ON PV"
  B3:11/2  "DP START MODE CHOSEN AND DP DELAY IS DONE OSR FOR ALM"
  B3:11/3  "DP START MODE CHOSEN AND DP DELAY IS DONE OSR FOR ALM"
  B3:11/4  "HI DP AND DP START MODE CHOSEN"
  B3:11/6  "VLV A HOME ALM OSR"
  B3:11/7  "VLV A HOME ALM OSR"
  B3:11/8  "VLV A HOME ALM SEAL"
  B3:11/9  "VLV B HOME ALM OSR"
  B3:11/10  "VLV B HOME ALM OSR"
  B3:11/11  "VLV B HOME ALM SEAL"
  B3:12/0  "REGN START MODE IS NOT DP BUT DP IS HI ALM OSR"
  B3:12/1  "REGN START MODE IS NOT DP BUT DP IS HI ALM OSR"
  B3:12/2  "REGN START MODE IS NOT DP BUT DP IS HI ALM SEAL"
  B3:12/8  "D FILT HI DP ALM SEAL"
  B3:12/9  "D FILT HI DP RESET BUTTON"
  B3:12/10  "E FILTER DP HI ALM OSR"
  B3:12/11  "E FILTER DP HI ALM OSR"
  B3:12/12  "E FILT HI DP"
  B3:12/13  "REGN START MODE IS NOT DP BUT DP IS HI ALM MSG"
  B3:12/14  "HI DP / NO DP START HORN"
  B9:2/4  "MANUAL CONTROL VISIBILITY BIT"
  B12:3/11  "B FORCE OPEN VALVE FV12B WHEN IN MANUAL"
  B12:3/12  "B FORCE OPEN VALVE FV13B WHEN IN MANUAL"
  B12:3/13  "B FORCE ON VALVE FV11B WHEN IN MANUAL"
  B12:3/14  "B FORCE OPEN VALVE FV14B WHEN IN MANUAL"
  B12:3/15  "B FORCE OPEN VALVE FV15B WHEN IN MANUAL"
  B13:0/3  "FILTER MEMORY OF SEQUENTIAL START REGN"
  B13:0/11  "FILTER SYSTEM START REGN DUE TO DP W/TIME OF DAY DELAY OSR"
  B13:2/1  "FILT B START REGN DUE TO DP W/TIME OF DAY DELAY OSR"
  B13:2/5  ALMBANNERCLOSEPB  "ALARM BANNER CLOSE BUTTTON"
  B13:2/7  "FILT B DP DELAY COUNTER DONE ALRM OSR"
  B13:2/8  "FILT B DP DELAY COUNTER DONE ALRM OSR"
  B13:2/9  "FILT B HIGH DP ALARM BANNER"
  B13:2/10  "FILT B HIGH DP SEAL FOR ALM"
  B13:2/13  "RESET FILT D SERVICE/REGN GALLON TOT ON A NEW SERVICE RUN"
  B13:2/14  "RESET FILT D SERVICE/REGN GALLON TOT ON A NEW SERVICE RUN"
  B13:3/5  "B DAYS LEFT DISPLAY FOR OIT IF INTERVAL START IS ENABLED"
  B13:3/11  "A FORCE ON RAW WATER INLET VALVE FV101A WHEN IN MANUAL"
  B13:3/12  "A FORCE OFF VALVE FV12A WHEN IN MANUAL"
  B13:3/13  "A FORCE OFF VALVE FV3A WHEN IN MANUAL"
  B13:3/14  "A FORCE OFF VALVE FV4A WHEN IN MANUAL"
  B13:3/15  "A FORCE OFF VALVE FV5A WHEN IN MANUAL"
  B13:4/0  "E BYPASS VALVE BV116 FORCE ON IN MANUAL MODE"
  B13:4/1  "COMMON BW INLET VALVE FORCE OFF VALVE FV115 WHEN IN MANUAL"
  B13:4/2  "B FORCE OFF VALVE FV12B WHEN IN MANUAL"
  B13:4/3  "B FORCE OFF VALVE FV3B WHEN IN MANUAL"
  B13:4/4  "B FORCE OFF VALVE FV4B WHEN IN MANUAL"
  B13:4/5  "B FORCE OFF VALVE FV5B WHEN IN MANUAL"
  B13:4/6  "RESET ALL FLOW TOTAL PB ON OIT"
  B13:4/15  "C FORCE OFF VALVE FV11C WHEN IN MANUAL"
  B13:5/9  "FILT D ADVANCE REGN PB OSR FROM OIT ONLY OSR"
  B13:5/10  "FILT D ADVANCE REGN PB OSR FROM OIT ONLY OSR"
  B13:6/5  "FILT D END REGN PB"
  B13:6/10  "C FORCE OFF VALVE FV12C WHEN IN MANUAL"
  B13:6/11  "D FORCE OFF VALVE FV11D WHEN IN MANUAL"
  B13:6/12  "D FORCE OFF VALVE FV12D WHEN IN MANUAL"
  B13:15/5  "UNIT A   FILTER SETTLE"
  B13:15/15  "FILT SEQUENTIAL REGN MEMORY START B AFTER A IS DONE"
  B13:16/5  "UNIT B   FILTER SETTLE"
  B21:0/7  "FILTER A DP WITH TIME OF DAY DELAY IMMED OSR START"
  B21:1/6  "OSR"
  B21:3/0  "FLOW SENSOR A PULS OSR"
  B21:3/1  "FLOW SENSOR A PULS OSR"
  B21:3/5  "FILT A RAW WATER INLET VALVE GRAPHIC DISPLAY"
  B21:3/6  "FILT A SERVICE OUTLET GRAPHIC DISPLAY"
  B21:3/7  "FILT A BW OUT GRAPHIC DISPLAY"
  B21:3/8  "FILT A RINSE OUT GRAPHIC DISPLAY"
  B21:4/1  "FILT A BW IN GRAPHIC DISPLAY"
  B22:3/0  "FLOW SENSOR B PULS OSR"
  B22:3/1  "FLOW SENSOR B PULS OSR"
  B22:3/3  "FILTER B REGN START BY TOTAL BATCH OR INTERVAL WITH TIME OF DAY DELAY OSR"
  B22:3/4  "FILTER B REGN START BY TOTAL BATCH OR INTERVAL WITH TIME OF DAY DELAY OSR"
  B22:3/5  "FILT B RAW INLET GRAPHIC DISPLAY"
  B22:3/6  "FILT B SERVICE OUTLET/BW INLET TO OTHER TANK GRAPHIC DISPLAY"
  B22:3/7  "FILT  B BW OUT GRAPHIC DISPLAY"
  B22:3/8  "FILT B RINSE OUT GRAPHIC DISPLAY"
  B22:4/1  "FILT B BW IN GRAPHIC DISPLAY"
  B23:0/0  CFILT_FR  "UNIT C FAST RINSE"
  B23:0/1  CFILT_OFFLINE  "C FORCED OFFLINE"
  B23:0/3  "FILT C DP STARTREGN MEM IN CASE OF REGN LO OR TREATED /BW SUPLYTANK NOT HI ENOUGH"
  B23:0/6  "C WENT INTO REGN DUE TO HI DP MEMORY SEAL"
  B23:0/7  "FILTER C DP WITH TIME OF DAY DELAY IMMED OSR START"
  B23:0/8  "FILTER C DP WITH TIME OF DAY DELAY IMMED OSR START"
  B23:0/9  "FILT C /ADVANCE REGN PB FROM OIT ONLY"
  B23:0/10  "FILT C ADVANCE REGN PB OSR FROM OIT ONLY OSR"
  B23:0/11  "FILT C ADVANCE REGN PB OSR FROM OIT ONLY OSR"
  B23:0/12  "FILT C ADVANCE REGN PB OSR FROM OIT ONLY"
  B23:0/13  CFILT_BW  "UNIT C  FILTER BACKWASH"
  B23:0/14  CFILT_SETTLE  "FILTER C IN SETTLE"
  B23:0/15  "FILT C RUN INTERVAL REGN START MEM.+ AND BW WASTETANK IS NOT LOW ENOUGH TO ACCEPT WASTE ALM OSR"
  B23:1/0  "FILT C DP AFTER LVL OR REGN LOCKOUT  TO AVOID TC START OF BOTH FILTER AT SAME TIME OSR"
  B23:1/1  "FILT C REGN START PB ONLY- NOT ADVANCE"
  B23:1/2  CFILT_PULSE  "UNIT C PULSE MASTER CTR"
  B23:1/3  "FILTER C REGN START TOTAL BATCH OR INTERVAL WITH TIME OF DAY DLYY-NO OTHER UNIT IN REGN OSR"
  B23:1/4  CFILT_SERVICE  "UNIT C  FILTER IN SERVICE"
  B23:1/5  "FILT C END REGN PB"
  B23:1/6  "RESET FILT C SERVICE/REGN GALLON TOT ON A NEW SERVICE RUN"
  B23:1/7  "UNIT C HIGH FLOW OSR"
  B23:1/8  "UNIT C HIGH FLOW OSR"
  B23:1/9  "UNIT C HIGH FLOW ALARM MSG"
  B23:1/10  "UNIT C HIGH FLOW ALARM FOR HORN"
  B23:1/11  "UNIT C LO FLOW OSR"
  B23:1/12  "UNIT C LO FLOW OSR"
  B23:1/13  "UNIT C LO FLOW ALARM MSG"
  B23:1/14  "UNIT C LO FLOW ALARM FOR HORN"
  B23:1/15  "FILT C RUN INTERVAL REGN START MEM.+ AND BW WASTETANK IS NOT LOW ENOUGH TO ACCEPT WASTE ALM OSR"
  B23:2/0  "FILT C DP START REGN MEMORY IN CASE OF REGN LO OR BW SUPPLYTANK NOT HI ENOUGH LVL LO OSR"
  B23:2/1  "FILT C DP START REGN MEMORY IN CASE OF REGN LO OR BW SUPPLYTANK NOT HI ENOUGH LVL LO OSR"
  B23:2/2  "UNIT C DP START REQUESTED AND TREATED WTR/BW SUPPLY TNK IS NOT HI ENOUGH ALM SEAL"
  B23:2/3  "UNIT C DP START REQUESTED AND BW SUPPLY TNK IS NOT HI ENOUGH ALM MSG"
  B23:2/4  "FILT C RUN INTERVAL REGN START MEM.+ AND BW WASTETANK IS NOT LOW ENOUGH TO ACCEPT WASTE ALMSEAL"
  B23:2/5  "FILT C DP STARTREGN MEM IN CASE OF WASTE NOT TANK LOW ENOUGH TO START BW"
  B23:2/6  "FILT C DP STARTREGN MEM IN CASE OF WASTE NOT TANK LOW ENOUGH TO START BW ALM OSR"
  B23:2/7  "FILT C DP STARTREGN MEM IN CASE OF WASTE NOT TANK LOW ENOUGH TO START BW ALM OSR"
  B23:2/8  "C BATCH REGN START MEMORY AND TREATED WATER/BW SUPPLY TANK IS HI OSR"
  B23:2/9  "C BATCH REGN START MEMORY AND TREATED WATER/BW SUPPLY TANK IS HI OSR"
  B23:2/10  "C BATCH REGN START MEM.TREATED/BW SUPPLY TANK IS NOT HI ENOUGH ALM BAN SEAL"
  B23:2/11  "C BATCH REGN START MEM.TREATED/BW SUPPLY TANK IS NOT HI ENOUGH ALM SEAL"
  B23:2/12  "FILT C RUN INTERVAL REGN START MEMORY AND BW SUPPLYTANK IS NOTHI ENOUGH OR REGN LOCKOUT OSR"
  B23:2/13  "FILT C RUN INTERVAL REGN START MEMORY AND BW SUPPLYTANK IS NOTHI ENOUGH OR REGN LOCKOUT OSR"
  B23:2/14  "C RUN TIME ELAPSED DONE START MEMORY AND BW TANK IS HI OR REGN LOCKOUT ALM MSG"
  B23:2/15  "FILT C RUN INTERVAL REGN START MEM.+TREA TED/BW SUPPLYTANK IS NOTHI ENOUGH OR REGN LO ALM HORN"
  B23:3/0  "FLOW SENSOR C PULS OSR"
  B23:3/1  "FLOW SENSOR C PULS OSR"
  B23:3/2  "RESET FILT C SERVICE/REGN GALLON TOT ON A NEW SERVICE RUN"
  B23:3/3  "FILTER C REGN START TOTAL BATCH OR INTERVAL WITH TIME OF DAY DELAY OSR"
  B23:3/4  "FILTER C REGN START TOTAL BATCH OR INTERVAL WITH TIME OF DAY DELAY OSR"
  B23:3/5  "FILT C RAW IN GRAPHIC DISPLAY"
  B23:3/6  "FILT C SERVICE OUTLET/BW INLET TO OTHER TANK GRAPHIC DISPLAY"
  B23:3/7  "FILT C BW OUT GRAPHIC DISPLAY"
  B23:3/8  "FILT C RINSE OUT GRAPHIC DISPLAY"
  B23:3/9  "UNIT C ONGOING SERVICE FLOW CTR IS GREATER THAN 1 MILLION OSR"
  B23:3/10  "UNIT C ONGOING SERVICE FLOW CTR IS GREATER THAN 1 MILLION OSR"
  B23:3/12  "C BATCH REGN START MEMORY& BW WASTE TANK IS NOT LO ENOUGH TO ACCEPT WASTE OSR FOR ALM"
  B23:3/13  "C BATCH REGN START MEMORY& BW WASTE TANK IS NOT LO ENOUGH TO ACCEPT WASTE OSR FOR ALM"
  B23:3/14  "C BATCH REGN START MEMORY& BW WASTE TANK IS NOT LO ENOUGH TO ACCEPT WASTE SEAL FOR ALM"
  B23:4/0  "FILT C DP STARTREGN MEM IN CASE OF WASTE NOT TANK LOW ENOUGH TO START BW ALM SEAL"
  B23:15/0  CARBAFILTREGN  "CARBON FILTER IN REGENERATION"
  B24:0/0  DFILT_FR  "UNIT D FAST RINSE"
  B24:0/1  DFILT_OFFLINE  "D FORCED OFFLINE"
  B24:0/3  "FILT D DP STARTREGN MEM IN CASE OF REGN LO OR TREATED /BW SUPLYTANK NOT HI ENOUGH"
  B24:0/4  "D BATCH REGN START MEMORY& TREATED/BW SUPPLY TANK IS NOT HI ENOUGH OR REGN LO"
  B24:0/5  "FILT D RUN INTERVAL REGNSTART MEMORY AND BW SUPPLY TANK IS NOT HI ENOUGH OR REGN LOCKOUT"
  B24:0/6  "D WENT INTO REGN DUE TO HI DP MEMORY SEAL"
  B24:0/7  "FILTER D DP WITH TIME OF DAY DELAY IMMED OSR START"
  B24:0/8  "FILTER D DP WITH TIME OF DAY DELAY IMMED OSR START"
  B24:0/9  "FILT D /ADVANCE REGN PB FROM OIT ONLY"
  B24:0/10  "FILT D ADVANCE REGN PB OSR FROM OIT ONLY OSR"
  B24:0/11  "FILT D ADVANCE REGN PB OSR FROM OIT ONLY OSR"
  B24:0/12  "FILT D ADVANCE REGN PB OSR FROM OIT ONLY"
  B24:0/13  DFILT_BW  "UNIT D IN BACKWASH"
  B24:0/14  DFILT_SETTLE  "UNIT D IN SETTLE"
  B24:1/0  "FILT D DP AFTER LVL OR REGN LOCKOUT  TO AVOID TC START OF BOTH FILTER AT SAME TIME OSR"
  B24:1/1  "FILT D REGN START PB ONLY- NOT ADVANCE"
  B24:1/2  DFILT_PULSE  "UNIT D PULSE MASTER CTR"
  B24:1/3  "FILTER D REGN START TOTAL BATCH OR INTERVAL WITH TIME OF DAY DLYY-NO OTHER UNIT IN REGN OSR"
  B24:1/4  DFILT_SERVICE  "UNIT D  FILTER IN SERVICE"
  B24:1/5  "FILT D END REGN PB"
  B24:1/7  "UNIT D HIGH FLOW OSR"
  B24:1/8  "UNIT D HIGH FLOW OSR"
  B24:1/9  "UNIT D HIGH FLOW ALARM MSG"
  B24:1/10  "UNIT D HIGH FLOW ALARM FOR HORN"
  B24:1/11  "UNIT D LO FLOW OSR"
  B24:1/12  "UNIT D LO FLOW OSR"
  B24:1/13  "UNIT D LO FLOW ALARM MSG"
  B24:1/14  "UNIT D LO FLOW ALARM FOR HORN"
  B24:2/5  "FILT D DP STARTREGN MEM IN CASE OF WASTE NOT TANK LOW ENOUGH TO START BW"
  B24:2/8  "D BATCH REGN START MEMORY AND TREATED WATER/BW SUPPLY TANK IS HI OSR"
  B24:2/9  "D BATCH REGN START MEMORY AND TREATED WATER/BW SUPPLY TANK IS HI OSR"
  B24:2/10  "D BATCH REGN START MEM.TREATED/BW SUPPLY TANK IS NOT HI ENOUGH ALM BAN SEAL"
  B24:2/11  "D BATCH REGN START MEM.TREATED/BW SUPPLY TANK IS NOT HI ENOUGH ALM SEAL"
  B24:2/12  "FILT D RUN INTERVAL REGNSTART MEMORY AND BW SUPPLY TANK IS NOT HI ENOUGH OR REGN LOCKOUT OSR"
  B24:2/13  "FILT D RUN INTERVAL REGNSTART MEMORY AND BW SUPPLY TANK IS NOT HI ENOUGH OR REGN LOCKOUT OSR"
  B24:2/14  "FILT D RUN INTERVAL REGNSTART MEMORY AND BW SUPPLY TANK IS NOT HI ENOUGH OR REGN LOCKOUT ALMMSG"
  B24:2/15  "FILT D RUN INTERVAL REGN START MEM.+TREA TED/BW SUPPLYTANK IS NOTHI ENOUGH OR REGN LO ALM HORN"
  B24:3/3  "FILTER D REGN START TOTAL BATCH OR INTERVAL WITH TIME OF DAY DELAY OSR"
  B24:3/4  "FILTER D REGN START TOTAL BATCH OR INTERVAL WITH TIME OF DAY DELAY OSR"
  B24:3/11  "D BATCH REGN START MEMORY& BW WASTE TANK IS NOT LO ENOUGH TO ACCEPT WASTE"
  B24:3/15  "FILT D RUN INTERVAL REGN START MEM.+ AND BW WASTETANK IS NOT LOW ENOUGH TO ACCEPT WASTE"
  C5:3  "FLOW SENSOR A PULS CTR"
  C5:5  "FLOW SENSOR B PULS CTR"
  C5:6  "FILTER C 60 MINUTE COUNTER FOR TIME INTERVAL"
  C5:16  "DUMP VALVE OPEN CTR PRE FROM N7:7"
  C5:21  "DUMP VALVE OPEN DELAY AFTER A FR PRESET FROM"
  C15:1  "FILTER B HOUR COUNTER FOR RUN INTERVAL LOGIC"
  C15:10  "FILTER B DP MINUTES CTR TO INITIATE REGN ENTRY FROM N17:15"
  F8:20  "TEMP # FOR PULSE MATH-PULSE DURATION/1000 ENTERED FROM N34:37"
  F8:21  "1/F8:20 PULSE MATH FOR FREQUENCY MATH"
  F8:48  "TEMP STORAGE OF A+B REGN WATER FLOW TOTAL FOR MATH FOR DISPLAY"
  F8:50  "TEMP ADD OF A+B ONGOING SER FLOW TOT FOR SYSTEM TOT THOUSANDS CALC"
  F8:52  "TEMP STORAGE OF A+B SERVICE AND REGN WATER FLOW TOTAL FOR MATH FOR DISPLAY"
  F8:61  "WELL PUMP HI LEVEL TURN OFF ENTRY"
  F8:62  "WELL PUMP ENABLE LEVEL ENTRY"
  F8:67  "GALLONS PER 1/10 SECOND FOR CHEMPUMP2 MATH"
  F8:68  "C GALLONS PER 1/10TH SECOND FOR PTO MATH"
  F8:69  "P2 LOGIC FOR CL TOTAL INLET GALL PER 1/10TH SECOND FOR CHEM PULSING A+B TEMP REGISTER"
  F8:71  "P-2 CL INLET TOTAL GALLONS FOR CHEM PACING"
  F8:72  "TEMP STORAGE OF A+B SERV ONGOING FLOW TOT MILLIONS FIELD"
  F8:78  "TEMP ADD OF A+B+C MILLIONS FIELD WHEN THOUS FIELD IS GRT 1 MILL AND LESS THAN 2 MILL"
  F8:83  "TEMP ADD OF A+B THOUSANDS FIELD"
  F8:84  "TEMP ADD OF A+B THOUSANDS FIELD"
  F8:85  "TEMP ADD A+B MILLIONS FIELD"
  F8:86  "TEMP ADD OF A+B MILLIONS FIELD"
  F8:87  "TEMP ADD OF A+B THOUS FIELD"
  F8:88  "TEMP STORAGE OF A+B THOUSANDS FIELD"
  F8:89  "GAL TOTAL ENTRY FROM PV TO STROKE PUMP"
  F8:91  "NAOCL LOGIC FOR TOTAL INLET GALL PER 1/10TH SECOND FOR CHEM PULSING A+B TEMP REGISTER"
  F8:92  "CHEMPUMP2 LOGIC FOR TOTAL INLET GALL PER 1/10TH SECOND FOR CHEM PULSING TEMP REGISTER"
  F8:93  "NAOH LOGIC FOR TOTAL INLET GALL PER 1/10TH SECOND FOR CHEM PULSING A+B TEMP REGISTER"
  F8:94  "POLYMER LOGIC FOR TOTAL INLET GALL PER 1/10TH SECOND FOR CHEM PULSING A+B TEMP REGISTER"
  F8:102  "CHEMPUMP2 GALLONS PER 1/10 SECOND TOTALIZER FOR PUMP PACING LOGIC"
  F8:103  "NAOH A+B GALLONS PER 1/10 SECOND TOTALIZER FOR NAOH PUMP PACING LOGIC"
  F8:104  "POLYMER A+B GALLONS PER 1/10 SECOND TOTALIZER FOR NAOH PUMP PACING LOGIC"
  F8:121  "GPM SETPOINT FOR CHEMPUMP1"
  F8:122  "GPM SETPOINT FOR CHEMPUMP2"
  F8:123  "GALLON TOTAL ENTRY FROM PV TO STROKE NAOH PUMP"
  F8:124  "NAOH A+B GALLONS PER 1/10 SECOND TOTALIZER FOR POLYMER PUMP PACING LOGIC"
  FILT_B_END_REGNPB  
  I:0.0/0  FE_101A_IN  "FLOW SENSOR A PULSE INPUT"
  I:0.0/1  "SPARE"
  I:0.0/2  "SPARE"
  I:0.0/3  "SPARE"
  I:0.0/4  FE_101B_IN  "FLOW SENSOR B PULSE INPUT"
  I:0.0/5  SPARE
  I:0.0/7  "SPARE"
  I:0.0/8  FE_101C_IN  "FLOW SENSOR C PULSE INPUT"
  I:0.0/9  "SPARE"
  I:0.0/10  "SPARE"
  I:1.0  "UNIT A FLOW 4-20=0-150GPM"
  I:1.0/13  DPS2  "FILT DP OPEN ON HIGH"
  I:1.1  "UNIT B FLOW 4-20=0-150GPM"
  N7:1  "HI FLOW DELAY ENTRY FOR ALM"
  N7:2  "LOW FLOW DELAY FOR ALARM"
  N7:3  "DUMP VALVE DELAY TO OPEN AFTER FR ENTRY FROM PV"
  N7:7  "DUMP VALVE OPEN PRESET FROM PV"
  N7:10  "BACKWASH RECYCLE/WASTE TANK LEVEL DISPLAY"
  N7:12  "DELAY IN MIN"
  N7:13  "MINUTES LEFT IN DUMP VALVE OPEN DISPLAY"
  N7:14  "DUMP VALVE AUTO MANUAL CONTROL SELEC 0=AUTO 1=MANUAL"
  N7:15  "FILTER A,B DP DELAY ENTRY IN MINUTES FROM OIT"
  N7:19  "MINUTES LEFT IN DELAY DISPLAY"
  N7:20  "DUMP VALVE HOA 0=AUTO 1=CLOSE 2=OPEN"
  N7:21  "014A STATUS"
  N7:24  "015A STATUS"
  N7:25  "011B STATUS"
  N7:26  "013B STATUS"
  N7:27  "012B STATUS"
  N7:28  "014B STATUS"
  N7:29  "015B STATUS"
  N7:30  "HORN STATUS"
  N7:31  "REGEN STATUS STATUS"
  N7:34  "BW STORAGE/RECYCLE TANK LVL LOW TO STOP ITS PUMP"
  N7:37  "CHEM PUMP2 STATUS 0=MAN 1=AUTO"
  N7:38  PT_100_IN_
  N7:39  PT_102_IN_
  N7:40  "PID AUTO.MANUAL MAINTAINED BUTTON 0=AUTO 1=MANUAL"
  N7:52  "PULSE OUTPUT LENGTH IN MILLISECS FOR CHEMPUMP2 PRESET"
  N7:61  "RESET TERM ENTRY FROM PV"
  N7:62  "RATE TERM ENTRY FROM PV"
  N17:0  "FILTER B DP DELAY LEFT IN MINUTES DISPLAY ON OIT"
  N17:3  "WEDNESDAY CHOICE FROM OIT 0=NO 1=CHOSEN"
  N17:7  "FRIDAY CHOICE FROM OIT 0=NO 1=CHOSEN"
  N17:9  "SATURDAY CHOICE FROM OIT 0=NO 1=CHOSEN"
  N17:20  "DAY OF THE WEEK FOR FILTER O-6=SUN-SAT"
  N34:9  "A+B GPM FOR MATH"
  N34:15  "REGEN TRIGGER ON DP FOR PV"
  N34:16  "REGEN TRIGGER ON VOL FOR PV"
  N34:17  "REGEN TRIGGER ON TIME FOR PV"
  N34:20  "BW PUMP HOA 1=HAND 0=OFF 2=AUTO"
  N34:27  "ENTRY FROM OIT TO ALLOW SETTLIN OF BW TANK BEFORE URNING BW PUMP"
  N34:34  "C VALVES AUTO/MANUAL CONTROL 0=AUTO 1=MANUAL"
  N34:37  "FILTER C HOUR OF DAY TO START SELECT EITHER DUE TO BATCH OR ELAPSED TIME OR DP"
  N34:38  "FILTER C MIN OF DAY TO START SELECT EITHER DUE TO BATCH OR ELAPSED TIME"
  N34:45  "FILTER B AUTO/MANUAL ADVANCE SELECT 0=AUTO 1=MANUAL"
  N34:46  "FILTER A TIME OF DAY TO START SELECT FOR BATCH START MODE"
  N34:47  "FILTER B TIME OF DAY TO START SELECT FOR BATCH START MODE"
  N34:50  C_MINUS_A
  N34:51  "C HRS LEFT TO REGEN"
  N34:52  "FILT A INTERVAL IN DAYS TO START A  REGN"
  N34:53  "C_DAYS_LEFT"
  N34:56  "FILTER C HOUR OF DAY TO START SELECT EITHER DUE TO BATCH OR ELAPSED TIME OR DP"
  N34:57  "FILTER C MIN OF DAY TO START SELECT EITHER DUE TO BATCH OR ELAPSED TIME"
  N34:64  "COMMON BW/FR IN VALVES AUTO/MANUAL CONTROL 0=AUTO 1=MANUAL"
  N34:66  "P2 CL PUMP DURATION OF PULSE ENTRY IN MILLSECONDS"
  N34:67  "P2 CL CHEMICAL FEED PUMP OFF AUTO SELECT 0=OFF 1=AUTO"
  N34:68  "HI DP AND REGN START IS NOT DP ALM ENABLE SELECT"
  N34:69  "COMM BW/FR IN CNTROL 0=AUTO 1=FORCE CLOSED 2=FORCE ON"
  N34:75  "FILT B VALVE 15B CONTROL 0=AUTO 1=FORCE CLOSED 2=FORCE ON"
  N34:79  "COMMON BACKWASH INLET AUTO/MANUAL CONTROL 0=AUTO 1=MANUAL"
  N34:81  "COMMON BW IN VLV BV115 CONTROL 0=AUTO 1=FORCE CLOSED 2=FORCE ON"
  N34:83  "WELL PUMP CONTROL 1=HAND 0=OFF 2=AUTO"
  O:0.0/11  "SPARE"
  O:0.0/13  "SPARE"
  O:0.0/14  "SPARE"
  O:0.0/15  "SPARE"
  O:2.0  "TOTALIZED FLOW RATE IN GPM OUTPUT TO SERVICE WATER INLET FEED THROTTLE VALVEFOR 4-20 CONTRO"
  O:2.0/0  "FILTER A REGN INLET VALVE FV11A ENG TO OPEN"
  O:2.0/1  "FILTER B REGN INLET VALVE FV12B"
  O:2.0/2  "FILTER C REGN INLET VALVE 12C -ENG TO OPEN"
  O:2.0/3  "FILTER REGN WATER INLET VALVE FV12D-ENG TO OPEN"
  O:3.0  "CO2 PROPORTINAL VALVE MORE CO2=LESS PH"
  PD9:0.0/1  "PID AUTO/MANUAL BIT 1=MANUAL 0=AUTO"
  PD9:0.2  "CO2SETPOINT TO MAINTAIN FOR CO2 FEED"
  PD9:0.7  "CO2 PID MAX ANALOG VALUE FOR NUMERIC RANGE 0-16363"
  PD9:0.8  "CO2 PID MIN ANALOG VALUE FOR NUMERIC RANGE 0-16363"
  PFILE:14  "D AND E ARE MANUAL F ILTERS"
  PFILE:15  "WASTE RECYCLE WATER BACK TO INLET"
  PFILE:17  "RG B TMP"
  PFILE:19  "RECYCLE"
  PTO:0.1/0  PTO
  T4:1  "DELAY BW FEED PUMP ON TILL THE BW INLET VALVE OPENS FIRST"
  T4:2  "FILT C FILTER 60 SECOND PULSER FOR RUN INTERVAL"
  T4:19  "LEVEL IN BW SUPPLY TANK FALLS BELOW PERMISSIVE BW START LEVEL-"
  T4:21  "PULSE OUTPUT LENGTH FOR NAOH PUMP PRESET FROM N7:53"
  T4:22  "TREATED WATER/BW SUPPLY STORAGE TANK HI LVL DELAY FOR ALM"
  T4:23  "PULSE OUTPUT LENGTH FOR POLYMER PUMP PRESET FROM N7:54"
  T4:24  "B DRIVE MULTIPORT VALVE TIMER"
  T4:25  "VALVE A HOMING DELAY FRO ALM"
  T4:29  "VALVE C DELAY IN BETWEEN PB ADVANCES TO ALLOW VALVE TO TURN"
  T4:30  "VALVE D DELAY IN BETWEEN PB ADVANCES TO ALLOW VALVE TO TURN"
  T4:31  "LEVEL OK TO RUN BW FEED PUMP DELAY"
  T4:32  "VALVE B HOMING DELAY FRO ALM"
  T4:33  "HI LEVEL STOP WELL PUMP DELAY"
  T4:34  "TREATED WATER STORAGE TANK/BW SUPPLY WATER AT WELL PUMP RE-START LEVEL SEAL"
  T4:35  "VALVE C HOMING DELAY FRO ALM"
  T4:36  "NOT IN DP START MODE FILTER SYSTEM DP DELAY ONE MINUTE TIMER"
  T4:43  "FILT B DP DELAY TO AVOID SIMUTANEOUS REGN STARTS DUE TO DP IF TC DLY =SAME TIMER"
  T4:49  "FILT B DELAY AFTER LOCKOUT TO AVOID DP START OF BOTH FILTER AT SAME TIME"
  T4:56  "DUMP VALVE DELAY IN SECONDS-ENTRY FROM PV N7:3"
  T4:57  "DUMP VALVE OPEN TIME PERIOD MINUTE PULSER"
  T4:62  "C5:16 DONE"

COMMENTS NOT ATTACHED TO A CURRENT RUNG
  N34:15: P-2 CL PUMP PTO PACING LOGIC
  N34:16: P1- KOH PUMP PTO LOGIC-IS NOT INITIALY BEING USED
  F8:103: NAOH CEHM PUMP 3
  F8:104: POLYMER CHEM PUMP 4

REVISION NOTES
  0: after ship revision- rev 4 added bw recycle pump can't run unless it has well pump running input also

DATA TABLE (non-zero values as saved)
DATA B3
% B3:0 % 0X0000 0X0001 0X2000 0X0005 0X0000 0X6000 0X0020 0X0000 0X0000 0X0001
% B3:10 % 0X5000 0X0001 0X0001 0X0001
DATA T4
% .PRE .ACC %
% T4:0 % 60 0
% T4:1 % 15 0
% T4:2 % 60 50
% T4:3 % 3 0
% T4:4 % 135 32
% T4:5 % 10 0
% T4:6 % 10 0
% T4:7 % 10 0
% T4:8 % 10 0
% T4:9 % 40 0
% T4:10 % 60 0
% T4:11 % 10 0
% T4:12 % 300 0
% T4:13 % 5 0
% T4:14 % 40 0
% T4:15 % 40 0
% T4:16 % 5 0
% T4:17 % 20 0
% T4:18 % 20 0
% T4:19 % 10 0
% T4:20 % 5 0
% T4:21 % 50 0
% T4:22 % 15 0
% T4:23 % 50 0
% T4:24 % 2 0
% T4:25 % 60 0
% T4:26 % 20 0
% T4:27 % 5 0
% T4:28 % 1 0
% T4:29 % 1 0
% T4:30 % 1 0
% T4:31 % 20 0
% T4:32 % 60 0
% T4:33 % 10 0
% T4:34 % 10 0
% T4:35 % 60 0
% T4:36 % 60 0
% T4:37 % 10 10
% T4:38 % 1200 0
% T4:39 % 10 10
% T4:40 % 2 0
% T4:41 % 2 0
% T4:42 % 100 34
% T4:43 % 3600 0
% T4:44 % 4 0
% T4:45 % 5 0
% T4:46 % 3 0
% T4:47 % 7 0
% T4:48 % 9 0
% T4:49 % 3 0
% T4:50 % 4 0
% T4:51 % 5 0
% T4:52 % 3 0
% T4:53 % 60 0
% T4:54 % 60 32
% T4:55 % 10 0
DATA C5
% .PRE .ACC %
% C5:0 % 60 7
% C5:1 % 10 0
% C5:2 % 96 0
% C5:3 % 1000 0
% C5:4 % 60 6
% C5:5 % 1000 0
% C5:6 % 60 8
% C5:7 % 96 0
% C5:8 % 30000 5
% C5:9 % 30000 1
% C5:10 % 96 2
% C5:11 % 3 0
% C5:12 % 3 1
DATA N7
% N7:0 % 568 19 18 5 10 0 2 1 0 0
% N7:10 % 0 95 12 30000 0 2 28 9 9 30000
% N7:20 % 0 0 6 1 0 10 20 999 0 0
% N7:30 % 0 100 20 20 10 0 1 2 4993 3200
% N7:40 % 0 5 1 80 20 12 0 1200 0 0
% N7:50 % 0 500
DATA F8
% F8:5 % -34.07938 0 0 -34.09031 10
% F8:10 % 0 0.01093292 0 78.7 10000
% F8:15 % 10000 10000 0.4955527 889.3606 172.7955
% F8:20 % 0.03 33.33334 0 0 0
% F8:25 % 78.7 78.7 0 730.2866 0
% F8:35 % 0 0 0 0 80
% F8:40 % 20 0 0 0 0
% F8:45 % 0 0 0 63.35838 0
% F8:50 % 2873.137 0 0 0 1000000
% F8:55 % 777314.6 1000000 0 10.5 0
% F8:60 % 10 9.5 8 0 2
% F8:70 % 100 0.7099996 0 0 8.657895
% F8:75 % 0.6 0 0 2 0
% F8:80 % 9.46875 1 -23.50302 1000014 1000014
% F8:85 % 0 0 0 0 10
% F8:95 % 14 14 0 0 0
% F8:105 % 12.6 2.3 0 0 0
% F8:115 % 0 0 34.22153 10 0.1312217
% F8:120 % -34.09031 4.1
DATA B9
% B9:0 % 0X4140 0X0017 0X0000
DATA C10
% .PRE .ACC %
% C10:0 % 3 0
% C10:1 % 30000 1
DATA B21
% B21:0 % 0X0000 0X0000 0X0000 0X01F1 0X8002 0X0000 0X0000
DATA B22
% B22:0 % 0X2004 0X0000 0X0000 0X01E1 0X0002 0X0000 0X0000
DATA N34
% N34:0 % 0 2 0 4 0 0 0 94 0 0
% N34:10 % 3 4 4 0 0 1 0 1 3 35
% N34:20 % 2 0 0 0 0 0 1 0 0 0
% N34:30 % 7 0 0 0 0 30 58 3 0 94
% N34:40 % 125 0 125 0 60 0 2 2 0 0
% N34:50 % 120 94 102 4 125 0 1000 1000 1 1
% N34:60 % 1 5 100 0 1 15 25 1 0 2
% N34:70 % 0 60 120 60 180 0 0 0 0 0
% N34:80 % 0 0 0 2 0 0 0 0 0 0
